// TIA Portal V20 export
TYPE "LER_typeUserDefine"
// stored: Access Published
   STRUCT
      "Bool" : Array[0..99] of Bool;
      "DInt" : Array[0..19] of DInt;
      LReal : Array[0..19] of LReal;
      "String" : Array[0..9] of String[30];
   END_STRUCT;
END_TYPE
